// TIA Portal V16 export
// export: Created 2021-09-08T12:46:15.2726003Z, ExportSetting WithDefaults, DisplayName Totally Integrated Automation Portal, DisplayVersion V16 Update 3, DisplayName TIA Portal Version Control Interface, DisplayVersion V16 Update 2, DisplayName TIA Portal Openness, DisplayVersion V16 Update 3, DisplayName TIA Portal Teamcenter Gateway, DisplayVersion V16, DisplayName STEP 7 Professional, DisplayVersion V16 Update 3, DisplayName STEP 7 Safety, DisplayVersion V16, DisplayName WinCC Advanced, DisplayVersion V16 Update 3
FUNCTION_BLOCK "AllPID"   // FB3, FBD
{ S7_Optimized_Access := 'TRUE' }
VERSION : 0.1
// stored: AutoNumber true, IsIECCheckEnabled false, IsRetainMemResEnabled false, MemoryReserve 100, SetENOAutomatically false, UDAEnableTagReadback false
   VAR
      P30x { S7_SetPoint := 'True'} : "PID_Pump2Pu1Fc";
      P120x { S7_SetPoint := 'True'} : "PID_Pump2Pu1Fc";
      P150x { S7_SetPoint := 'True'} : "PID_Pump2Pu1Fc";
      P901 { S7_SetPoint := 'True'} : "PID_Pump";
      P1301 { S7_SetPoint := 'True'} : "PID_Pump";
   END_VAR
BEGIN

REGION Network 1: P30x
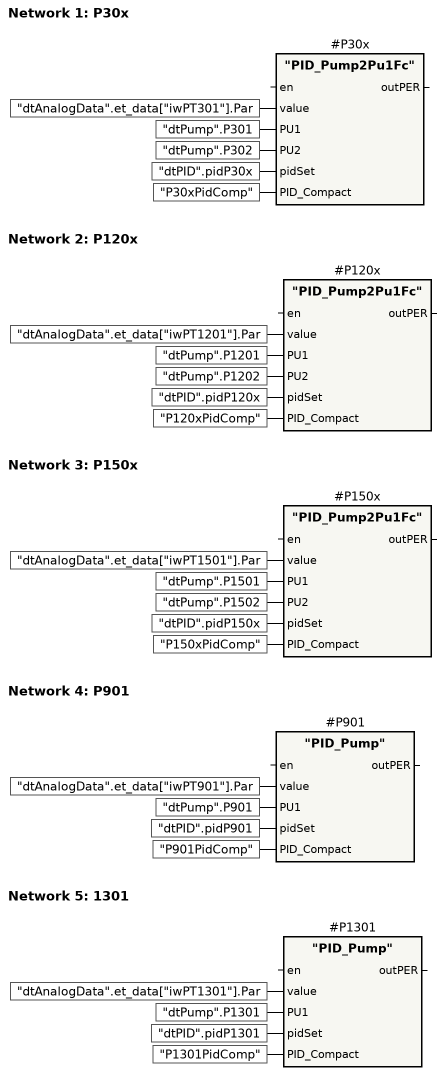
   #P30x(value := "dtAnalogData".et_data["iwPT301"].Par,   // "PID_Pump2Pu1Fc"
         PU1 := "dtPump".P301,
         PU2 := "dtPump".P302,
         pidSet := "dtPID".pidP30x,
         PID_Compact := "P30xPidComp");
END_REGION

REGION Network 2: P120x
   #P120x(value := "dtAnalogData".et_data["iwPT1201"].Par,   // "PID_Pump2Pu1Fc"
          PU1 := "dtPump".P1201,
          PU2 := "dtPump".P1202,
          pidSet := "dtPID".pidP120x,
          PID_Compact := "P120xPidComp");
END_REGION

REGION Network 3: P150x
   #P150x(value := "dtAnalogData".et_data["iwPT1501"].Par,   // "PID_Pump2Pu1Fc"
          PU1 := "dtPump".P1501,
          PU2 := "dtPump".P1502,
          pidSet := "dtPID".pidP150x,
          PID_Compact := "P150xPidComp");
END_REGION

REGION Network 4: P901
   #P901(value := "dtAnalogData".et_data["iwPT901"].Par,   // "PID_Pump"
         PU1 := "dtPump".P901,
         pidSet := "dtPID".pidP901,
         PID_Compact := "P901PidComp");
END_REGION

REGION Network 5: 1301
   #P1301(value := "dtAnalogData".et_data["iwPT1301"].Par,   // "PID_Pump"
          PU1 := "dtPump".P1301,
          pidSet := "dtPID".pidP1301,
          PID_Compact := "P1301PidComp");
END_REGION
END_FUNCTION_BLOCK
